// This function has been automatically generated from the project information.
{attribute 'signature_flag' := '1073741824'}
{attribute 'TcGenerated'}
{attribute 'no-analysis'}
FUNCTION F_GetVersion : ST_LibVersion
VAR_INPUT
	
END_VAR

F_GetVersion.iMajor := 0;
F_GetVersion.iMinor := 0;
F_GetVersion.iBuild := 4;
F_GetVersion.iRevision := 0;
F_GetVersion.sVersion := '0.0.4';
F_GetVersion.nFlags := 0;

END_FUNCTION

(* stored: Version 1.1.0.1, ProductVersion 3.1.4026.18
   POU F_GetVersion: Id {2326c2f6-493e-47a7-ad11-f8f79cf72f92}, SpecialFunc None *)
